KUKA KRL data list: p01drop3.dat

&ACCESS RVP1
&REL 48
&COMMENT drop carton
&PARAM EDITMASK = *
&PARAM TEMPLATE = C:\KRC\Roboter\Template\vorgabe
&PARAM DISKPATH = KRC:\R1\Program\Sub Programs
DEFDAT  p01drop3

EXT  BAS (BAS_COMMAND  :IN,REAL  :IN )
DECL INT SUCCESS
;******************************
;*     E6POS Declarations     *
;******************************

DECL E6POS XP01WAITREQ2={X 2157.35596,Y -301.755188,Z 2852.14893,A -15.8183,B 72.8074417,C -9.82211304,S 2,T 34,E1 0.0,E2 0.0,E3 0.0,E4 0.0,E5 0.0,E6 0.0}
DECL E6POS XP10={X 2411.43896,Y 1748.73096,Z -1095.62903,A -177.692307,B -16.9195194,C 42.7874298,S 2,T 34,E1 0.0,E2 0.0,E3 0.0,E4 0.0,E5 0.0,E6 0.0}
DECL E6POS XP20={X 1670.59900,Y -157.831207,Z 2354.64209,A -15.8183,B 72.8074417,C -9.82211304,S 2,T 34,E1 0.0,E2 0.0,E3 0.0,E4 0.0,E5 0.0,E6 0.0}
DECL E6POS XP30={X 1670.59900,Y -157.831207,Z 2354.64209,A -15.8183,B 72.8074417,C -9.82211304,S 2,T 34,E1 0.0,E2 0.0,E3 0.0,E4 0.0,E5 0.0,E6 0.0}
DECL E6POS XDROP_POS={X 1670.59900,Y -157.831207,Z 2354.64209,A -15.8183,B 72.8074417,C -9.82211304,S 2,T 34,E1 0.0,E2 0.0,E3 0.0,E4 0.0,E5 0.0,E6 0.0}
DECL E6POS XP40={X 2411.43896,Y 1748.73096,Z -1095.62903,A -177.692307,B -16.9195194,C 42.7874298,S 2,T 34,E1 0.0,E2 0.0,E3 0.0,E4 0.0,E5 0.0,E6 0.0}
DECL E6POS XP50={X 2411.43896,Y 1748.73096,Z -1095.62903,A -177.692307,B -16.9195194,C 42.7874298,S 2,T 34,E1 0.0,E2 0.0,E3 0.0,E4 0.0,E5 0.0,E6 0.0}
DECL E6POS XP01WAITREL2={X 2411.43896,Y 1748.73096,Z -1095.62903,A -177.692307,B -16.9195194,C 42.7874298,S 2,T 34,E1 0.0,E2 0.0,E3 0.0,E4 0.0,E5 0.0,E6 0.0}

;******************************
;*     FDAT Declarations      *
;******************************

DECL FDAT FP01WAITREQ2={TOOL_NO 12,BASE_NO 0,IPO_FRAME #BASE}
DECL FDAT FP10={TOOL_NO 12,BASE_NO 0,IPO_FRAME #TCP}
DECL FDAT FP20={TOOL_NO 12,BASE_NO 0,IPO_FRAME #TCP}
DECL FDAT FP30={TOOL_NO 12,BASE_NO 0,IPO_FRAME #TCP}
DECL FDAT FDROP_POS={TOOL_NO 12,BASE_NO 0,IPO_FRAME #TCP}
DECL FDAT FP40={TOOL_NO 12,BASE_NO 0,IPO_FRAME #TCP}
DECL FDAT FP50={TOOL_NO 12,BASE_NO 0,IPO_FRAME #TCP}
DECL FDAT FP01WAITREL2={TOOL_NO 12,BASE_NO 0,IPO_FRAME #TCP}

;******************************
;*  PDAT & LDAT Declarations  *
;******************************

DECL PDAT PH={VEL 100.000,ACC 100.000,APO_DIST 100.000,APO_MODE #CDIS,GEAR_JERK 100.000,EXAX_IGN 0}

DECL MODULEPARAM_T LAST_TP_PARAMS={PARAMS[] "FORDTECH.P_AREA_REQ=3; FORDTECH.P_SAFETY_POS=0; FORDTECH.P_RET=0; Kuka.VelocityFieldEnabled=True; Kuka.ColDetectFieldEnabled=True; Kuka.MovementParameterFieldEnabled=True; Kuka.IsAngleEnabled=False; Kuka.PointName=preDROPpoint; Kuka.FrameData.base_no=0; Kuka.FrameData.tool_no=5; Kuka.FrameData.ipo_frame=#BASE; Kuka.isglobalpoint=False; Kuka.MoveDataPtpName=H; Kuka.MovementDataPdat.apo_mode=#CDIS; Kuka.MovementDataPdat.apo_dist=100; Kuka.MovementData.vel=2; Kuka.MovementData.acc=100; Kuka.MovementData.exax_ign=0; Kuka.VelocityPtp=100; Kuka.BlendingEnabled=True; Kuka.APXEnabled=False; Kuka.CurrentCDSetIndex=0; Kuka.FrameData.point2=; FORDTECH.P_JOB_RDY=3; FORDTECH.P_AREA_REL=3; Kuka.MoveDataName=CPDAT2; Kuka.MovementData.cb={AUX_PT {ORI #CONSIDER,E1 #CONSIDER,E2 #CONSIDER,E3 #CONSIDER,E4 #CONSIDER,E5 #CONSIDER,E6 #CONSIDER},TARGET_PT {ORI #INTERPOLATE,E1 #INTERPOLATE,E2 #INTERPOLATE,E3 #INTERPOLATE,E4 #INTERPOLATE,E5 #INTERPOLATE,E6 #INTERPOLATE}}; Kuka.MovementData.apo_fac=50; Kuka.MovementData.apo_dist=500; Kuka.MovementData.axis_acc=100; Kuka.MovementData.axis_vel=100; Kuka.MovementData.circ_typ=#BASE; Kuka.MovementData.jerk_fac=50; Kuka.MovementData.ori_typ=#VAR; Kuka.VelocityPath=2       "}
DECL E6POS XP01Waitdrop={X 290.951508,Y 816.177185,Z 1155.55042,A -86.9976196,B 22.0779018,C -179.006119,S 6,T 27,E1 0.0,E2 0.0,E3 0.0,E4 0.0,E5 0.0,E6 0.0}
DECL FDAT FP01Waitdrop={TOOL_NO 5,BASE_NO 0,IPO_FRAME #BASE,POINT2[] " ",TQ_STATE FALSE}
DECL E6POS XBATPOS1={X 290.951233,Y 816.177124,Z 1155.55042,A -86.9976196,B 22.0779018,C -179.006119,S 6,T 27,E1 0.0,E2 0.0,E3 0.0,E4 0.0,E5 0.0,E6 0.0}
DECL FDAT FBATPOS1={TOOL_NO 5,BASE_NO 11,IPO_FRAME #BASE,POINT2[] " "}
DECL E6POS XBATPOS2={X 763.140686,Y 824.200684,Z 1155.55042,A -86.9976196,B 22.0779018,C -179.006119,S 6,T 27,E1 0.0,E2 0.0,E3 0.0,E4 0.0,E5 0.0,E6 0.0}
DECL FDAT FBATPOS2={TOOL_NO 5,BASE_NO 11,IPO_FRAME #BASE,POINT2[] " "}
DECL E6POS XBATPOS3={X 290.951263,Y 1017.51129,Z 1155.55042,A -86.9976196,B 22.0779018,C -179.006119,S 6,T 27,E1 0.0,E2 0.0,E3 0.0,E4 0.0,E5 0.0,E6 0.0}
DECL FDAT FBATPOS3={TOOL_NO 5,BASE_NO 11,IPO_FRAME #BASE,POINT2[] " "}
DECL E6POS XBATPOS4={X 768.407043,Y 1017.51129,Z 1155.55042,A -86.9976196,B 22.0779018,C -179.006119,S 6,T 27,E1 0.0,E2 0.0,E3 0.0,E4 0.0,E5 0.0,E6 0.0}
DECL FDAT FBATPOS4={TOOL_NO 5,BASE_NO 11,IPO_FRAME #BASE,POINT2[] " "}
DECL E6POS XBATPOS5={X 290.951263,Y 1218.65857,Z 1155.55042,A -86.9976196,B 22.0779018,C -179.006119,S 6,T 27,E1 0.0,E2 0.0,E3 0.0,E4 0.0,E5 0.0,E6 0.0}
DECL FDAT FBATPOS5={TOOL_NO 5,BASE_NO 11,IPO_FRAME #BASE,POINT2[] " "}
DECL E6POS XBATPOS6={X 738.674316,Y 1202.54663,Z 1155.55042,A -86.9976196,B 22.0779018,C -179.006119,S 6,T 27,E1 0.0,E2 0.0,E3 0.0,E4 0.0,E5 0.0,E6 0.0}
DECL FDAT FBATPOS6={TOOL_NO 5,BASE_NO 11,IPO_FRAME #BASE,POINT2[] " "}
DECL E6POS XBATPOS7={X 290.951263,Y 1386.78320,Z 1155.55042,A -86.9976196,B 22.0779018,C -179.006119,S 6,T 27,E1 0.0,E2 0.0,E3 0.0,E4 0.0,E5 0.0,E6 0.0}
DECL FDAT FBATPOS7={TOOL_NO 5,BASE_NO 11,IPO_FRAME #BASE,POINT2[] " "}
DECL E6POS XBATPOS8={X 728.249,Y 1368.06873,Z 1155.55042,A -86.9976196,B 22.0779018,C -179.006119,S 6,T 27,E1 0.0,E2 0.0,E3 0.0,E4 0.0,E5 0.0,E6 0.0}
DECL FDAT FBATPOS8={TOOL_NO 5,BASE_NO 11,IPO_FRAME #BASE,POINT2[] " "}
DECL E6POS XBATPOS9={X 290.951263,Y 1572.31165,Z 1155.55042,A -86.9976196,B 22.0779018,C -179.006119,S 6,T 27,E1 0.0,E2 0.0,E3 0.0,E4 0.0,E5 0.0,E6 0.0}
DECL FDAT FBATPOS9={TOOL_NO 5,BASE_NO 11,IPO_FRAME #BASE,POINT2[] " "}
DECL E6POS XBATPOS10={X 753.970337,Y 1583.41736,Z 1155.55042,A -86.9976196,B 22.0779018,C -179.006119,S 6,T 27,E1 0.0,E2 0.0,E3 0.0,E4 0.0,E5 0.0,E6 0.0}
DECL FDAT FBATPOS10={TOOL_NO 5,BASE_NO 11,IPO_FRAME #BASE,POINT2[] " "}
DECL E6POS XBATPOS11={X 301.951050,Y 1774.17639,Z 1155.55042,A -86.9976196,B 22.0779018,C -179.006119,S 6,T 27,E1 0.0,E2 0.0,E3 0.0,E4 0.0,E5 0.0,E6 0.0}
DECL FDAT FBATPOS11={TOOL_NO 5,BASE_NO 11,IPO_FRAME #BASE,POINT2[] " "}
DECL E6POS XBATPOS12={X 738.848694,Y 1774.17639,Z 1155.55042,A -86.9976196,B 22.0779018,C -179.006119,S 6,T 27,E1 0.0,E2 0.0,E3 0.0,E4 0.0,E5 0.0,E6 0.0}
DECL FDAT FBATPOS12={TOOL_NO 5,BASE_NO 11,IPO_FRAME #BASE,POINT2[] " "}
DECL E6POS XBATPOS13={X 442.124359,Y -682.465210,Z 1416.05603,A -171.206314,B 14.8656197,C -154.747955,S 6,T 26,E1 0.0,E2 0.0,E3 0.0,E4 0.0,E5 0.0,E6 0.0}
DECL FDAT FBATPOS13={TOOL_NO 5,BASE_NO 0,IPO_FRAME #BASE,POINT2[] " ",TQ_STATE FALSE}
DECL E6POS XDROPpoint={X 471.147,Y -1067.04773,Z 1223.22400,A -179.451859,B -0.162765205,C 179.769058,S 6,T 26,E1 0.0,E2 0.0,E3 0.0,E4 0.0,E5 0.0,E6 0.0}
DECL FDAT FDROPpoint={TOOL_NO 5,BASE_NO 0,IPO_FRAME #BASE,POINT2[] " ",TQ_STATE FALSE}
DECL LDAT LCPDAT1={VEL 2.00000,ACC 100.000,APO_DIST 500.000,APO_FAC 50.0000,AXIS_VEL 100.000,AXIS_ACC 100.000,ORI_TYP #VAR,CIRC_TYP #BASE,JERK_FAC 50.0000,GEAR_JERK 100.000,EXAX_IGN 0,CB {AUX_PT {ORI #CONSIDER,E1 #CONSIDER,E2 #CONSIDER,E3 #CONSIDER,E4 #CONSIDER,E5 #CONSIDER,E6 #CONSIDER},TARGET_PT {ORI #INTERPOLATE,E1 #INTERPOLATE,E2 #INTERPOLATE,E3 #INTERPOLATE,E4 #INTERPOLATE,E5 #INTERPOLATE,E6 #INTERPOLATE}}}
DECL E6POS XpreDROPpoint={X 471.147,Y -1067.04773,Z 1308.08960,A -179.451859,B -0.162765205,C 179.769058,S 6,T 26,E1 0.0,E2 0.0,E3 0.0,E4 0.0,E5 0.0,E6 0.0}
DECL FDAT FpreDROPpoint={TOOL_NO 5,BASE_NO 0,IPO_FRAME #BASE,POINT2[] " ",TQ_STATE FALSE}
DECL LDAT LCPDAT2={VEL 2.00000,ACC 100.000,APO_DIST 500.000,APO_FAC 50.0000,AXIS_VEL 100.000,AXIS_ACC 100.000,ORI_TYP #VAR,CIRC_TYP #BASE,JERK_FAC 50.0000,GEAR_JERK 100.000,EXAX_IGN 0,CB {AUX_PT {ORI #CONSIDER,E1 #CONSIDER,E2 #CONSIDER,E3 #CONSIDER,E4 #CONSIDER,E5 #CONSIDER,E6 #CONSIDER},TARGET_PT {ORI #INTERPOLATE,E1 #INTERPOLATE,E2 #INTERPOLATE,E3 #INTERPOLATE,E4 #INTERPOLATE,E5 #INTERPOLATE,E6 #INTERPOLATE}}}
DECL E6POS XBATPOS14={X 442.124359,Y -682.465210,Z 1416.05603,A -171.206314,B 14.8656197,C -154.747955,S 6,T 26,E1 0.0,E2 0.0,E3 0.0,E4 0.0,E5 0.0,E6 0.0}
DECL FDAT FBATPOS14={TOOL_NO 5,BASE_NO 11,IPO_FRAME #BASE,POINT2[] " ",TQ_STATE FALSE}
DECL BASIS_SUGG_T LAST_BASIS={POINT1[] "P45                     ",POINT2[] "P45                     ",CP_PARAMS[] "CPDAT0                  ",PTP_PARAMS[] "PDAT24                  ",CONT[] "                        ",CP_VEL[] "2.0                     ",PTP_VEL[] "100                     ",SYNC_PARAMS[] "SYNCDAT                 ",SPL_NAME[] "S0                      ",A_PARAMS[] "ADAT0                   "}
DECL PDAT PPDAT1={VEL 100.000,ACC 100.000,APO_DIST 100.000,GEAR_JERK 50.0000,EXAX_IGN 0}
DECL PDAT PPDAT2={VEL 100.000,ACC 100.000,APO_DIST 100.000,GEAR_JERK 50.0000,EXAX_IGN 0}
DECL PDAT PPDAT3={VEL 100.000,ACC 100.000,APO_DIST 100.000,GEAR_JERK 50.0000,EXAX_IGN 0}
DECL PDAT PPDAT4={VEL 100.000,ACC 100.000,APO_DIST 100.000,GEAR_JERK 50.0000,EXAX_IGN 0}
DECL PDAT PPDAT5={VEL 100.000,ACC 100.000,APO_DIST 100.000,APO_MODE #CDIS,GEAR_JERK 50.0000,EXAX_IGN 0}
DECL LDAT LCPDAT3={VEL 2.00000,ACC 100.000,APO_DIST 100.000,APO_FAC 50.0000,AXIS_VEL 100.000,AXIS_ACC 100.000,ORI_TYP #VAR,CIRC_TYP #BASE,JERK_FAC 50.0000,GEAR_JERK 50.0000,EXAX_IGN 0}
DECL LDAT LCPDAT4={VEL 2.00000,ACC 100.000,APO_DIST 100.000,APO_FAC 50.0000,AXIS_VEL 100.000,AXIS_ACC 100.000,ORI_TYP #VAR,CIRC_TYP #BASE,JERK_FAC 50.0000,GEAR_JERK 50.0000,EXAX_IGN 0}
DECL E6POS XP1={X 716.539490,Y -339.002350,Z 1261.05945,A -151.411957,B 9.54572201,C -170.760315,S 6,T 26,E1 0.0,E2 0.0,E3 0.0,E4 0.0,E5 0.0,E6 0.0}
DECL FDAT FP1={TOOL_NO 5,BASE_NO 0,IPO_FRAME #BASE,POINT2[] " ",TQ_STATE FALSE}
DECL PDAT PPDAT6={VEL 100.000,ACC 100.000,APO_DIST 100.000,APO_MODE #CDIS,GEAR_JERK 50.0000,EXAX_IGN 0}
DECL E6POS XP2={X 629.440857,Y 383.904541,Z 1179.93518,A -112.750427,B 20.1261520,C -170.604736,S 6,T 27,E1 0.0,E2 0.0,E3 0.0,E4 0.0,E5 0.0,E6 0.0}
DECL FDAT FP2={TOOL_NO 5,BASE_NO 0,IPO_FRAME #BASE,POINT2[] " ",TQ_STATE FALSE}
DECL PDAT PPDAT7={VEL 100.000,ACC 100.000,APO_DIST 100.000,APO_MODE #CDIS,GEAR_JERK 50.0000,EXAX_IGN 0}
DECL E6POS XP3={X -532.723450,Y 1638.84937,Z 2302.56665,A -87.9836655,B 0.794596434,C 91.2849731,S 6,T 27,E1 0.0,E2 0.0,E3 0.0,E4 0.0,E5 0.0,E6 0.0}
DECL FDAT FP3={TOOL_NO 5,BASE_NO 0,IPO_FRAME #BASE,POINT2[] " ",TQ_STATE FALSE}
DECL PDAT PPDAT8={VEL 100.000,ACC 100.000,APO_DIST 100.000,APO_MODE #CDIS,GEAR_JERK 50.0000,EXAX_IGN 0}
DECL E6POS XP4={X -1118.90833,Y 1713.72119,Z 2268.47095,A -88.1086884,B 0.787056804,C 91.3148880,S 6,T 27,E1 0.0,E2 0.0,E3 0.0,E4 0.0,E5 0.0,E6 0.0}
DECL FDAT FP4={TOOL_NO 5,BASE_NO 0,IPO_FRAME #BASE,POINT2[] " ",TQ_STATE FALSE}
DECL LDAT LCPDAT5={VEL 2.00000,ACC 100.000,APO_DIST 10.0000,APO_FAC 50.0000,AXIS_VEL 100.000,AXIS_ACC 100.000,ORI_TYP #VAR,CIRC_TYP #BASE,JERK_FAC 50.0000,GEAR_JERK 50.0000,EXAX_IGN 0}
DECL E6POS XP5={X -1770.77356,Y 1828.03650,Z 2007.82544,A -88.1926193,B 0.862227559,C 88.8579407,S 6,T 27,E1 0.0,E2 0.0,E3 0.0,E4 0.0,E5 0.0,E6 0.0}
DECL FDAT FP5={TOOL_NO 5,BASE_NO 0,IPO_FRAME #BASE,POINT2[] " ",TQ_STATE FALSE}
DECL LDAT LCPDAT6={VEL 2.00000,ACC 100.000,APO_DIST 100.000,APO_FAC 50.0000,AXIS_VEL 100.000,AXIS_ACC 100.000,ORI_TYP #VAR,CIRC_TYP #BASE,JERK_FAC 50.0000,GEAR_JERK 50.0000,EXAX_IGN 0}
DECL E6POS XP6={X -1745.08875,Y 1731.76428,Z 2190.31567,A -87.5496750,B 1.31373835,C 86.8927383,S 6,T 27,E1 0.0,E2 0.0,E3 0.0,E4 0.0,E5 0.0,E6 0.0}
DECL FDAT FP6={TOOL_NO 5,BASE_NO 0,IPO_FRAME #BASE,POINT2[] " ",TQ_STATE FALSE}
DECL LDAT LCPDAT7={VEL 2.00000,ACC 100.000,APO_DIST 100.000,APO_FAC 50.0000,AXIS_VEL 100.000,AXIS_ACC 100.000,ORI_TYP #VAR,CIRC_TYP #BASE,JERK_FAC 50.0000,GEAR_JERK 50.0000,EXAX_IGN 0}
DECL E6POS XP7={X -1697.77173,Y 1754.19934,Z 2222.69678,A -88.2045746,B 0.886862755,C 88.0748,S 6,T 27,E1 0.0,E2 0.0,E3 0.0,E4 0.0,E5 0.0,E6 0.0}
DECL FDAT FP7={TOOL_NO 5,BASE_NO 0,IPO_FRAME #BASE,POINT2[] " ",TQ_STATE FALSE}
DECL PDAT PPDAT9={VEL 100.000,ACC 100.000,APO_DIST 100.000,APO_MODE #CDIS,GEAR_JERK 50.0000,EXAX_IGN 0}
DECL E6POS XP8={X -1686.30774,Y 1828.03613,Z 2203.44702,A -88.1479797,B 0.813352,C 90.4450073,S 6,T 27,E1 0.0,E2 0.0,E3 0.0,E4 0.0,E5 0.0,E6 0.0}
DECL FDAT FP8={TOOL_NO 5,BASE_NO 0,IPO_FRAME #BASE,POINT2[] " ",TQ_STATE FALSE}
DECL PDAT PPDAT10={VEL 100.000,ACC 100.000,APO_DIST 100.000,APO_MODE #CDIS,GEAR_JERK 50.0000,EXAX_IGN 0}
DECL E6POS XP9={X -1686.30774,Y 1828.03613,Z 1755.45349,A -88.1479797,B 0.813352168,C 90.4450073,S 6,T 27,E1 0.0,E2 0.0,E3 0.0,E4 0.0,E5 0.0,E6 0.0}
DECL FDAT FP9={TOOL_NO 5,BASE_NO 0,IPO_FRAME #BASE,POINT2[] " ",TQ_STATE FALSE}
DECL LDAT LCPDAT8={VEL 2.00000,ACC 100.000,APO_DIST 100.000,APO_FAC 50.0000,AXIS_VEL 100.000,AXIS_ACC 100.000,ORI_TYP #VAR,CIRC_TYP #BASE,JERK_FAC 50.0000,GEAR_JERK 50.0000,EXAX_IGN 0}
DECL E6POS XP11={X -1420.73376,Y 573.312378,Z 2220.34766,A -76.5273361,B -0.934734046,C 87.5865,S 6,T 27,E1 0.0,E2 0.0,E3 0.0,E4 0.0,E5 0.0,E6 0.0}
DECL FDAT FP11={TOOL_NO 5,BASE_NO 0,IPO_FRAME #BASE,POINT2[] " ",TQ_STATE FALSE}
DECL LDAT LCPDAT9={VEL 2.00000,ACC 100.000,APO_DIST 100.000,APO_FAC 50.0000,AXIS_VEL 100.000,AXIS_ACC 100.000,ORI_TYP #VAR,CIRC_TYP #BASE,JERK_FAC 50.0000,GEAR_JERK 50.0000,EXAX_IGN 0}
DECL E6POS XP12={X -1731.80762,Y 1731.76428,Z 2212.77319,A -87.5575104,B 1.32822061,C 86.5535889,S 6,T 27,E1 0.0,E2 0.0,E3 0.0,E4 0.0,E5 0.0,E6 0.0}
DECL FDAT FP12={TOOL_NO 5,BASE_NO 0,IPO_FRAME #BASE,POINT2[] " ",TQ_STATE FALSE}
DECL LDAT LCPDAT10={VEL 2.00000,ACC 100.000,APO_DIST 100.000,APO_FAC 50.0000,AXIS_VEL 100.000,AXIS_ACC 100.000,ORI_TYP #VAR,CIRC_TYP #BASE,JERK_FAC 50.0000,GEAR_JERK 50.0000,EXAX_IGN 0}
DECL E6POS XP13={X -1343.92920,Y 1963.01379,Z 1625.04541,A -89.1568909,B 0.804959893,C 90.4484558,S 6,T 27,E1 0.0,E2 0.0,E3 0.0,E4 0.0,E5 0.0,E6 0.0}
DECL FDAT FP13={TOOL_NO 5,BASE_NO 0,IPO_FRAME #BASE,POINT2[] " ",TQ_STATE FALSE}
DECL LDAT LCPDAT11={VEL 2.00000,ACC 100.000,APO_DIST 100.000,APO_FAC 50.0000,AXIS_VEL 100.000,AXIS_ACC 100.000,ORI_TYP #VAR,CIRC_TYP #BASE,JERK_FAC 50.0000,GEAR_JERK 50.0000,EXAX_IGN 0}
DECL LDAT LCPDAT0={VEL 2.00000,ACC 100.000,APO_DIST 10.0000,APO_FAC 50.0000,AXIS_VEL 100.000,AXIS_ACC 100.000,ORI_TYP #VAR,CIRC_TYP #BASE,JERK_FAC 50.0000,GEAR_JERK 50.0000,EXAX_IGN 0}
DECL E6POS XP0={X -142.561630,Y 1779.97058,Z 1596.68616,A -89.4406509,B 9.14810,C -179.615814,S 6,T 27,E1 0.0,E2 0.0,E3 0.0,E4 0.0,E5 0.0,E6 0.0}
DECL FDAT FP0={TOOL_NO 5,BASE_NO 0,IPO_FRAME #BASE,POINT2[] " ",TQ_STATE FALSE}
DECL LDAT LCPDAT12={VEL 2.00000,ACC 100.000,APO_DIST 100.000,APO_FAC 50.0000,AXIS_VEL 100.000,AXIS_ACC 100.000,ORI_TYP #VAR,CIRC_TYP #BASE,JERK_FAC 50.0000,GEAR_JERK 50.0000,EXAX_IGN 0}
DECL E6POS XP14={X -1696.23901,Y 1932.78906,Z 1444.85730,A -88.9868927,B 0.802531540,C 90.6850204,S 6,T 27,E1 0.0,E2 0.0,E3 0.0,E4 0.0,E5 0.0,E6 0.0}
DECL FDAT FP14={TOOL_NO 5,BASE_NO 0,IPO_FRAME #BASE,POINT2[] " ",TQ_STATE FALSE}
DECL LDAT LCPDAT13={VEL 2.00000,ACC 100.000,APO_DIST 100.000,APO_FAC 50.0000,AXIS_VEL 100.000,AXIS_ACC 100.000,ORI_TYP #VAR,CIRC_TYP #BASE,JERK_FAC 50.0000,GEAR_JERK 50.0000,EXAX_IGN 0}
DECL E6POS XP15={X -916.910156,Y 1788.28918,Z 1596.68604,A -89.4406509,B 9.14809608,C -179.615814,S 6,T 27,E1 0.0,E2 0.0,E3 0.0,E4 0.0,E5 0.0,E6 0.0}
DECL FDAT FP15={TOOL_NO 5,BASE_NO 0,IPO_FRAME #BASE,POINT2[] " ",TQ_STATE FALSE}
DECL E6POS XP16={X -1503.82495,Y 558.656,Z 1628.41663,A -75.1206360,B -0.934732616,C 87.5864944,S 6,T 27,E1 0.0,E2 0.0,E3 0.0,E4 0.0,E5 0.0,E6 0.0}
DECL FDAT FP16={TOOL_NO 5,BASE_NO 0,IPO_FRAME #BASE,POINT2[] " ",TQ_STATE FALSE}
DECL LDAT LCPDAT14={VEL 2.00000,ACC 100.000,APO_DIST 100.000,APO_FAC 50.0000,AXIS_VEL 100.000,AXIS_ACC 100.000,ORI_TYP #VAR,CIRC_TYP #BASE,JERK_FAC 50.0000,GEAR_JERK 50.0000,EXAX_IGN 0}
DECL PDAT PPDAT11={VEL 100.000,ACC 100.000,APO_DIST 100.000,APO_MODE #CDIS,GEAR_JERK 50.0000,EXAX_IGN 0}
DECL PDAT PPDAT12={VEL 100.000,ACC 100.000,APO_DIST 100.000,APO_MODE #CDIS,GEAR_JERK 50.0000,EXAX_IGN 0}
DECL E6POS XP17={X -1157.21924,Y 879.505859,Z 2231.63,A -75.1206360,B -0.934732735,C 87.5864944,S 6,T 27,E1 0.0,E2 0.0,E3 0.0,E4 0.0,E5 0.0,E6 0.0}
DECL FDAT FP17={TOOL_NO 5,BASE_NO 0,IPO_FRAME #BASE,POINT2[] " ",TQ_STATE FALSE}
DECL PDAT PPDAT13={VEL 100.000,ACC 100.000,APO_DIST 100.000,APO_MODE #CDIS,GEAR_JERK 50.0000,EXAX_IGN 0}
DECL PDAT PPDAT14={VEL 100.000,ACC 100.000,APO_DIST 100.000,APO_MODE #CDIS,GEAR_JERK 50.0000,EXAX_IGN 0}
DECL E6POS XP18={X -142.561630,Y 1779.97058,Z 1596.68616,A -89.4406509,B 9.14810,C -179.615814,S 6,T 27,E1 0.0,E2 0.0,E3 0.0,E4 0.0,E5 0.0,E6 0.0}
DECL FDAT FP18={TOOL_NO 5,BASE_NO 0,IPO_FRAME #BASE,POINT2[] " ",TQ_STATE FALSE}
DECL LDAT LCPDAT15={VEL 2.00000,ACC 100.000,APO_DIST 100.000,APO_FAC 50.0000,AXIS_VEL 100.000,AXIS_ACC 100.000,ORI_TYP #VAR,CIRC_TYP #BASE,JERK_FAC 50.0000,GEAR_JERK 50.0000,EXAX_IGN 0}
DECL E6POS XP19={X 445.718170,Y 1685.51,Z 1387.29028,A -89.2562790,B 3.86068535,C 177.573654,S 6,T 27,E1 0.0,E2 0.0,E3 0.0,E4 0.0,E5 0.0,E6 0.0}
DECL FDAT FP19={TOOL_NO 5,BASE_NO 0,IPO_FRAME #BASE,POINT2[] " ",TQ_STATE FALSE}
DECL LDAT LCPDAT16={VEL 2.00000,ACC 100.000,APO_DIST 100.000,APO_FAC 50.0000,AXIS_VEL 100.000,AXIS_ACC 100.000,ORI_TYP #VAR,CIRC_TYP #BASE,JERK_FAC 50.0000,GEAR_JERK 50.0000,EXAX_IGN 0}
DECL E6POS XP21={X 544.058960,Y 1724.54578,Z 1005.91003,A -89.3502274,B -0.653226912,C -179.937820,S 6,T 27,E1 0.0,E2 0.0,E3 0.0,E4 0.0,E5 0.0,E6 0.0}
DECL FDAT FP21={TOOL_NO 5,BASE_NO 0,IPO_FRAME #BASE,POINT2[] " ",TQ_STATE FALSE}
DECL LDAT LCPDAT17={VEL 2.00000,ACC 100.000,APO_DIST 100.000,APO_FAC 50.0000,AXIS_VEL 100.000,AXIS_ACC 100.000,ORI_TYP #VAR,CIRC_TYP #BASE,JERK_FAC 50.0000,GEAR_JERK 50.0000,EXAX_IGN 0}
DECL E6POS XP22={X 445.718170,Y 1685.51,Z 1387.29028,A -89.2562790,B 3.86068535,C 177.573654,S 6,T 27,E1 0.0,E2 0.0,E3 0.0,E4 0.0,E5 0.0,E6 0.0}
DECL FDAT FP22={TOOL_NO 5,BASE_NO 0,IPO_FRAME #BASE,POINT2[] " ",TQ_STATE FALSE}
DECL PDAT PPDAT15={VEL 100.000,ACC 100.000,APO_DIST 100.000,APO_MODE #CDIS,GEAR_JERK 50.0000,EXAX_IGN 0}
DECL E6POS XP23={X -1553.22266,Y 1713.72131,Z 2268.47095,A -88.1086884,B 0.786908329,C 91.3148804,S 6,T 27,E1 0.0,E2 0.0,E3 0.0,E4 0.0,E5 0.0,E6 0.0}
DECL FDAT FP23={TOOL_NO 5,BASE_NO 0,IPO_FRAME #BASE,POINT2[] " ",TQ_STATE FALSE}
DECL PDAT PPDAT16={VEL 100.000,ACC 100.000,APO_DIST 100.000,APO_MODE #CDIS,GEAR_JERK 50.0000,EXAX_IGN 0}
DECL E6POS XP24={X -1580.58740,Y 1929.36243,Z 2203.94092,A -89.8538513,B 0.163948148,C 88.5617447,S 6,T 27,E1 0.0,E2 0.0,E3 0.0,E4 0.0,E5 0.0,E6 0.0}
DECL FDAT FP24={TOOL_NO 5,BASE_NO 0,IPO_FRAME #BASE,POINT2[] " ",TQ_STATE FALSE}
DECL LDAT LCPDAT18={VEL 2.00000,ACC 100.000,APO_DIST 100.000,APO_FAC 50.0000,AXIS_VEL 100.000,AXIS_ACC 100.000,ORI_TYP #VAR,CIRC_TYP #BASE,JERK_FAC 50.0000,GEAR_JERK 50.0000,EXAX_IGN 0}
DECL E6POS XP25={X -1578.04492,Y 1929.36243,Z 1618.60583,A -90.1842270,B 0.163948819,C 88.5617447,S 6,T 27,E1 0.0,E2 0.0,E3 0.0,E4 0.0,E5 0.0,E6 0.0}
DECL FDAT FP25={TOOL_NO 5,BASE_NO 0,IPO_FRAME #BASE,POINT2[] " ",TQ_STATE FALSE}
DECL LDAT LCPDAT19={VEL 2.00000,ACC 100.000,APO_DIST 100.000,APO_FAC 50.0000,AXIS_VEL 100.000,AXIS_ACC 100.000,ORI_TYP #VAR,CIRC_TYP #BASE,JERK_FAC 50.0000,GEAR_JERK 50.0000,EXAX_IGN 0}
DECL E6POS XP26={X -1364.34216,Y 1929.36243,Z 1812.72021,A -89.4744,B 0.176458865,C 90.6702576,S 6,T 27,E1 0.0,E2 0.0,E3 0.0,E4 0.0,E5 0.0,E6 0.0}
DECL FDAT FP26={TOOL_NO 5,BASE_NO 0,IPO_FRAME #BASE,POINT2[] " ",TQ_STATE FALSE}
DECL E6POS XP27={X -916.910156,Y 1788.28918,Z 1596.68604,A -89.4406509,B 9.14809608,C -179.615814,S 6,T 27,E1 0.0,E2 0.0,E3 0.0,E4 0.0,E5 0.0,E6 0.0}
DECL FDAT FP27={TOOL_NO 5,BASE_NO 0,IPO_FRAME #BASE,POINT2[] " ",TQ_STATE FALSE}
DECL LDAT LCPDAT20={VEL 2.00000,ACC 100.000,APO_DIST 100.000,APO_FAC 50.0000,AXIS_VEL 100.000,AXIS_ACC 100.000,ORI_TYP #VAR,CIRC_TYP #BASE,JERK_FAC 50.0000,GEAR_JERK 50.0000,EXAX_IGN 0}
DECL E6POS XP28={X -1420.73376,Y 573.312378,Z 1621.20483,A -76.5273361,B -0.934734046,C 87.5865,S 6,T 27,E1 0.0,E2 0.0,E3 0.0,E4 0.0,E5 0.0,E6 0.0}
DECL FDAT FP28={TOOL_NO 5,BASE_NO 0,IPO_FRAME #BASE,POINT2[] " ",TQ_STATE FALSE}
DECL LDAT LCPDAT21={VEL 2.00000,ACC 100.000,APO_DIST 100.000,APO_FAC 50.0000,AXIS_VEL 100.000,AXIS_ACC 100.000,ORI_TYP #VAR,CIRC_TYP #BASE,JERK_FAC 50.0000,GEAR_JERK 50.0000,EXAX_IGN 0}
DECL E6POS XP29={X -1513.85889,Y 1963.01379,Z 1513.09802,A -89.1568909,B 0.804959834,C 90.4484558,S 6,T 27,E1 0.0,E2 0.0,E3 0.0,E4 0.0,E5 0.0,E6 0.0}
DECL FDAT FP29={TOOL_NO 5,BASE_NO 0,IPO_FRAME #BASE,POINT2[] " ",TQ_STATE FALSE}
DECL LDAT LCPDAT22={VEL 2.00000,ACC 100.000,APO_DIST 100.000,APO_FAC 50.0000,AXIS_VEL 100.000,AXIS_ACC 100.000,ORI_TYP #VAR,CIRC_TYP #BASE,JERK_FAC 50.0000,GEAR_JERK 50.0000,EXAX_IGN 0}
DECL E6POS XP31={X -1553.64111,Y 1962.81079,Z 1512.98438,A -89.1568909,B 0.804959893,C 90.4484558,S 6,T 27,E1 0.0,E2 0.0,E3 0.0,E4 0.0,E5 0.0,E6 0.0}
DECL FDAT FP31={TOOL_NO 5,BASE_NO 0,IPO_FRAME #BASE,POINT2[] " ",TQ_STATE FALSE}
DECL LDAT LCPDAT23={VEL 2.00000,ACC 100.000,APO_DIST 100.000,APO_FAC 50.0000,AXIS_VEL 100.000,AXIS_ACC 100.000,ORI_TYP #VAR,CIRC_TYP #BASE,JERK_FAC 50.0000,GEAR_JERK 50.0000,EXAX_IGN 0}
DECL E6POS XP32={X -1691.51086,Y 1853.95801,Z 2214.78296,A -89.9661942,B 0.122944221,C 90.4054108,S 6,T 27,E1 0.0,E2 0.0,E3 0.0,E4 0.0,E5 0.0,E6 0.0}
DECL FDAT FP32={TOOL_NO 5,BASE_NO 0,IPO_FRAME #BASE,POINT2[] " ",TQ_STATE FALSE}
DECL LDAT LCPDAT24={VEL 2.00000,ACC 100.000,APO_DIST 100.000,APO_FAC 50.0000,AXIS_VEL 100.000,AXIS_ACC 100.000,ORI_TYP #VAR,CIRC_TYP #BASE,JERK_FAC 50.0000,GEAR_JERK 50.0000,EXAX_IGN 0}
DECL E6POS XP33={X -1691.51086,Y 1942.26245,Z 1609.76379,A -89.9661942,B 0.122944236,C 90.4054108,S 6,T 27,E1 0.0,E2 0.0,E3 0.0,E4 0.0,E5 0.0,E6 0.0}
DECL FDAT FP33={TOOL_NO 5,BASE_NO 0,IPO_FRAME #BASE,POINT2[] " ",TQ_STATE FALSE}
DECL LDAT LCPDAT25={VEL 2.00000,ACC 100.000,APO_DIST 100.000,APO_FAC 50.0000,AXIS_VEL 100.000,AXIS_ACC 100.000,ORI_TYP #VAR,CIRC_TYP #BASE,JERK_FAC 50.0000,GEAR_JERK 50.0000,EXAX_IGN 0}
DECL E6POS XP34={X -955.242126,Y 1693.14233,Z 1131.74048,A -90.8804550,B -0.952020586,C 177.437790,S 6,T 27,E1 0.0,E2 0.0,E3 0.0,E4 0.0,E5 0.0,E6 0.0}
DECL FDAT FP34={TOOL_NO 5,BASE_NO 0,IPO_FRAME #BASE,POINT2[] " ",TQ_STATE FALSE}
DECL LDAT LCPDAT26={VEL 2.00000,ACC 100.000,APO_DIST 100.000,APO_FAC 50.0000,AXIS_VEL 100.000,AXIS_ACC 100.000,ORI_TYP #VAR,CIRC_TYP #BASE,JERK_FAC 50.0000,GEAR_JERK 50.0000,EXAX_IGN 0}
DECL E6POS XP35={X -1673.92334,Y 1936.45679,Z 1857.99097,A -89.8400497,B -1.45816052,C 88.5053406,S 6,T 27,E1 0.0,E2 0.0,E3 0.0,E4 0.0,E5 0.0,E6 0.0}
DECL FDAT FP35={TOOL_NO 5,BASE_NO 0,IPO_FRAME #BASE,POINT2[] " ",TQ_STATE FALSE}
DECL LDAT LCPDAT27={VEL 2.00000,ACC 100.000,APO_DIST 100.000,APO_FAC 50.0000,AXIS_VEL 100.000,AXIS_ACC 100.000,ORI_TYP #VAR,CIRC_TYP #BASE,JERK_FAC 50.0000,GEAR_JERK 50.0000,EXAX_IGN 0}
DECL E6POS XSAIDA={X -1593.17566,Y 1927.33374,Z 1408.19226,A -89.4182358,B 0.822354257,C 89.0936279,S 6,T 27,E1 0.0,E2 0.0,E3 0.0,E4 0.0,E5 0.0,E6 0.0}
DECL FDAT Fsaida={TOOL_NO 5,BASE_NO 0,IPO_FRAME #BASE,POINT2[] " ",TQ_STATE FALSE}
DECL LDAT LCPDAT28={VEL 2.00000,ACC 100.000,APO_DIST 100.000,APO_FAC 50.0000,AXIS_VEL 100.000,AXIS_ACC 100.000,ORI_TYP #VAR,CIRC_TYP #BASE,JERK_FAC 50.0000,GEAR_JERK 50.0000,EXAX_IGN 0}
DECL LDAT LCPDAT29={VEL 2.00000,ACC 100.000,APO_DIST 100.000,APO_FAC 50.0000,AXIS_VEL 100.000,AXIS_ACC 100.000,ORI_TYP #VAR,CIRC_TYP #BASE,JERK_FAC 50.0000,GEAR_JERK 50.0000,EXAX_IGN 0}
DECL E6POS XP36={X -1593.17566,Y 1927.33374,Z 1408.19226,A -89.4182358,B 0.822354317,C 89.0936279,S 6,T 27,E1 0.0,E2 0.0,E3 0.0,E4 0.0,E5 0.0,E6 0.0}
DECL FDAT FP36={TOOL_NO 5,BASE_NO 0,IPO_FRAME #BASE,POINT2[] " ",TQ_STATE FALSE}
DECL E6POS XP28SALI={X -1586.92261,Y 1926.27112,Z 1486.64294,A -89.4182358,B 0.822354317,C 89.0936279,S 6,T 27,E1 0.0,E2 0.0,E3 0.0,E4 0.0,E5 0.0,E6 0.0}
DECL FDAT FP28sali={TOOL_NO 5,BASE_NO 0,IPO_FRAME #BASE,POINT2[] " ",TQ_STATE FALSE}
DECL E6POS XP37={X -142.561630,Y 1779.97058,Z 1596.68616,A -89.4406509,B 9.14810,C -179.615814,S 6,T 27,E1 0.0,E2 0.0,E3 0.0,E4 0.0,E5 0.0,E6 0.0}
DECL FDAT FP37={TOOL_NO 5,BASE_NO 0,IPO_FRAME #BASE,POINT2[] " ",TQ_STATE FALSE}
DECL PDAT PPDAT17={VEL 100.000,ACC 100.000,APO_DIST 100.000,APO_MODE #CDIS,GEAR_JERK 50.0000,EXAX_IGN 0}
DECL E6POS XP38={X -142.561630,Y 1779.97058,Z 1596.68616,A -89.4406509,B 9.14810,C -179.615814,S 6,T 27,E1 0.0,E2 0.0,E3 0.0,E4 0.0,E5 0.0,E6 0.0}
DECL FDAT FP38={TOOL_NO 5,BASE_NO 0,IPO_FRAME #BASE,POINT2[] " ",TQ_STATE FALSE}
DECL PDAT PPDAT18={VEL 100.000,ACC 100.000,APO_DIST 100.000,APO_MODE #CDIS,GEAR_JERK 50.0000,EXAX_IGN 0}
DECL E6POS XP39={X -955.242126,Y 1693.14233,Z 1081.74048,A -90.8804550,B -0.952020526,C 177.437790,S 6,T 27,E1 0.0,E2 0.0,E3 0.0,E4 0.0,E5 0.0,E6 0.0}
DECL FDAT FP39={TOOL_NO 5,BASE_NO 0,IPO_FRAME #BASE,POINT2[] " ",TQ_STATE FALSE}
DECL PDAT PPDAT19={VEL 100.000,ACC 100.000,APO_DIST 100.000,GEAR_JERK 50.0000,EXAX_IGN 0}
DECL E6POS XP41={X -956.779724,Y 1694.71301,Z 830.002258,A -90.8889618,B -0.888903737,C 178.570831,S 6,T 27,E1 0.0,E2 0.0,E3 0.0,E4 0.0,E5 0.0,E6 0.0}
DECL FDAT FP41={TOOL_NO 5,BASE_NO 0,IPO_FRAME #BASE,POINT2[] " ",TQ_STATE FALSE}
DECL PDAT PPDAT20={VEL 100.000,ACC 100.000,APO_DIST 100.000,GEAR_JERK 50.0000,EXAX_IGN 0}
DECL E6POS XP42={X -952.557373,Y 1735.80811,Z 838.628479,A -90.8710938,B -0.906417727,C 177.430542,S 6,T 27,E1 0.0,E2 0.0,E3 0.0,E4 0.0,E5 0.0,E6 0.0}
DECL FDAT FP42={TOOL_NO 5,BASE_NO 0,IPO_FRAME #BASE,POINT2[] " ",TQ_STATE FALSE}
DECL PDAT PPDAT21={VEL 100.000,ACC 100.000,APO_DIST 100.000,GEAR_JERK 50.0000,EXAX_IGN 0}
DECL E6POS XP43={X 565.289795,Y 1726.80969,Z 950.139709,A -89.3770676,B -2.01419520,C -179.295013,S 6,T 27,E1 0.0,E2 0.0,E3 0.0,E4 0.0,E5 0.0,E6 0.0}
DECL FDAT FP43={TOOL_NO 5,BASE_NO 0,IPO_FRAME #BASE,POINT2[] " ",TQ_STATE FALSE}
DECL PDAT PPDAT22={VEL 100.000,ACC 100.000,APO_DIST 100.000,GEAR_JERK 50.0000,EXAX_IGN 0}
DECL E6POS XP44={X 565.289795,Y 1701.06067,Z 830.396606,A -89.2956696,B -0.384512693,C 178.381790,S 6,T 27,E1 0.0,E2 0.0,E3 0.0,E4 0.0,E5 0.0,E6 0.0}
DECL FDAT FP44={TOOL_NO 5,BASE_NO 0,IPO_FRAME #BASE,POINT2[] " ",TQ_STATE FALSE}
DECL PDAT PPDAT23={VEL 100.000,ACC 100.000,APO_DIST 100.000,GEAR_JERK 50.0000,EXAX_IGN 0}
DECL E6POS XP45={X 578.367065,Y 1726.80969,Z 793.225708,A -89.4170532,B 0.609481633,C 178.789703,S 6,T 27,E1 0.0,E2 0.0,E3 0.0,E4 0.0,E5 0.0,E6 0.0}
DECL FDAT FP45={TOOL_NO 5,BASE_NO 0,IPO_FRAME #BASE,POINT2[] " ",TQ_STATE FALSE}
DECL PDAT PPDAT24={VEL 100.000,ACC 100.000,APO_DIST 100.000,GEAR_JERK 50.0000,EXAX_IGN 0}
ENDDAT
